PROGRAM P_Serial_Com
VAR
	fbSerialLineControl_EL6001_P1: SerialLineControl;
	fbSerialLineControl_EL6001_P2: SerialLineControl;
	fbSerialLineControl_EL6001_P3: SerialLineControl;
END_VAR

//These are the global IOs...don't forget to copy your data into them

(* EL6001 Serial port 0 com function *)
fbSerialLineControl_EL6001_P1(
	Mode:= SERIALLINEMODE_EL6_22B (*SERIALLINEMODE_KL6_22B_STANDARD*),
	pComIn:= ADR(Serial_P1_stComIn),
	pComOut:=ADR(Serial_P1_stComOut) ,
	SizeComIn:= SIZEOF(Serial_P1_stComIn),
	TxBuffer:= Serial_P1_SerialTXBuffer,
	RxBuffer:= Serial_P1_SerialRXBuffer,
	Error=> ,
	ErrorID=> );
fbSerialLineControl_EL6001_P2(
	Mode:= SERIALLINEMODE_EL6_22B (*SERIALLINEMODE_KL6_22B_STANDARD*),
	pComIn:= ADR(Serial_P2_stComIn),
	pComOut:=ADR(Serial_P2_stComOut) ,
	SizeComIn:= SIZEOF(Serial_P2_stComIn),
	TxBuffer:= Serial_P2_SerialTXBuffer,
	RxBuffer:= Serial_P2_SerialRXBuffer,
	Error=> ,
	ErrorID=> );
fbSerialLineControl_EL6001_P3(
	Mode:= SERIALLINEMODE_EL6_22B (*SERIALLINEMODE_KL6_22B_STANDARD*),
	pComIn:= ADR(Serial_P3_stComIn),
	pComOut:=ADR(Serial_P3_stComOut) ,
	SizeComIn:= SIZEOF(Serial_P3_stComIn),
	TxBuffer:= Serial_P3_SerialTXBuffer,
	RxBuffer:= Serial_P3_SerialRXBuffer,
	Error=> ,
	ErrorID=> );

END_PROGRAM

(* stored: Version 1.1.0.1, ProductVersion 3.1.4020.12
   POU P_Serial_Com: Id {fa981f30-4d2c-4d48-ab6c-00ec78d696a1}, SpecialFunc None *)
